	122:	(* manual down *)
		MD := TRUE;
		MU := FALSE;
		IF POS <= EXT_TRIG THEN
			(* extend cycle if bottom is reached *)
			POS := BYTE#0;
			last := tx;
			STATUS := BYTE#129;	(* extend *)
		END_IF;

	123:	(* auto positioning *)
		MD := rmp.DN;
		MU := rmp.UP;
		IF NOT (rmp.DN OR rmp.UP) THEN
			(* automatic position is reached *)
			IF POS <= EXT_TRIG THEN
				(* extend at bottom *)
				MD := TRUE;
				last := tx;
				STATUS := BYTE#129;	(* extend *)
			ELSIF POS >= USINT_TO_BYTE(USINT#255 - BYTE_TO_USINT(EXT_TRIG)) THEN
				(* extend at top *)
				MU := TRUE;
				last := tx;
				STATUS := BYTE#129;	(* extend *)
			ELSE
				STATUS := S_IN;
			END_IF;
		END_IF;

	124:	(* revert from top or bottom *)
		MD := rmp.DN;
		MU := rmp.UP;
		IF NOT(rmp.DN OR rmp.UP) THEN
(*		IF POS = rmp.IN THEN  *)
			PI_last := PI;
			STATUS := S_IN;
		END_IF;

	127:	(* lockout time *)
		IF (tx - last) >= T_LOCKOUT THEN
				STATUS := S_IN;
		END_IF;

	128:	(* calibration *)
		MU := TRUE;
		MD := FALSE;
		rmp.IN := BYTE#255;
		IF (tx - last) >= (T_UP +  T_EXT) THEN
			MU := FALSE;
			last := tx;
			STATUS := BYTE#127;	(* lockout *)
		END_IF;

	129: (* extend mode *)
		IF (tx - last) >= T_EXT THEN
			MU := FALSE;
			MD := FALSE;
			last := tx;
			STATUS := BYTE#127;	(* lockout *)
		END_IF;

ELSE
	MU := FALSE;
	MD := FALSE;
	IF PI <> PI_last THEN
		PI_last := PI;
		rmp.IN := PI;
		STATUS := BYTE#123;	(* auto positioning *)
	ELSIF POS = BYTE#0 AND RU THEN
		rmp.IN := R_POS_BOT;
		STATUS := BYTE#124;	(* revert *)
	ELSIF pos = BYTE#255 AND RD THEN
		rmp.IN := R_POS_TOP;
		STATUS := BYTE#124;	(* revert *)
	ELSE
		STATUS := S_IN;
	END_IF;
END_CASE;

(* From OSCAT LIBRARY, www.oscat.de *)
(* T_PLC_MS, _RMP_NEXT required *)
          
END_FUNCTION_BLOCK

FUNCTION_BLOCK BLIND_INPUT
  VAR_INPUT
    POS : BYTE;
    ANG : BYTE;
    S1 : BOOL;
    S2 : BOOL;
    IN : BOOL;
    PI : BYTE;
    AI : BYTE;
    SINGLE_SWITCH : BOOL;
    CLICK_EN : BOOL := TRUE;
    CLICK_TIME : TIME := t#500ms;
    MAX_RUNTIME : TIME := t#60s;
    MANUAL_TIMEOUT : TIME := t#1h;
    DEBOUNCE_TIME : TIME := t#20ms;
    DBL_CLK1 : BOOL := FALSE;
    DBL_POS1 : BYTE;
    DBL_ANG1 : BYTE;
    DBL_CLK2 : BOOL := FALSE;
    DBL_POS2 : BYTE := 255;
    DBL_ANG2 : BYTE := 255;
    D1_TOGGLE : BOOL := TRUE;
    D2_TOGGLE : BOOL := TRUE;
    MASTER_MODE : BOOL;
  END_VAR
  VAR_OUTPUT
    QU : BOOL := TRUE;
    QD : BOOL := TRUE;
    STATUS : BYTE;
    PO : BYTE := 255;
    AO : BYTE := 255;
    D1 : BOOL;
    D2 : BOOL;
  END_VAR
  VAR
    s1e : TOF;
    s2e : TOF;
    s1d : CLICK_MODE;
    s2d : CLICK_MODE;
    dir : BOOL;
    tx : TIME;
    last : TIME;
  END_VAR

            tx:= UDINT_TO_TIME(T_PLC_MS(en:=true));

(* inputs S1 and S2 are debounced and then decoded for multiple clicks *)
s1e(in := S1, pt := DEBOUNCE_TIME);
s2e(in := S2, pt := DEBOUNCE_TIME);
s1d(in := (s1e.Q AND NOT SINGLE_SWITCH) OR (s1e.Q AND SINGLE_SWITCH AND dir), t_long := CLICK_TIME);
s2d(in := (s2e.Q AND NOT SINGLE_SWITCH) OR (s1e.Q AND SINGLE_SWITCH AND NOT dir), t_long := CLICK_TIME);

(* if d1 and d2 are not toggle clear them to make sure they are only active for oine cycle *)
IF NOT d1_toggle THEN d1 := FALSE; END_IF;
IF NOT d2_toggle THEN d2 := FALSE; END_IF;

(* decode actions *)
IF (s1d.LONG AND s2d.LONG) OR (status = BYTE#139) THEN
   status := BYTE#139;
   IF NOT (s1d.LONG OR s2d.LONG)  THEN status := BYTE#130; END_IF;
ELSIF s1d.tp_LONG THEN
	status := BYTE#132;
ELSIF s2d.tp_LONG THEN
	status := BYTE#133;
ELSIF  s1d.SINGLE THEN
	IF click_en THEN
		(* if running then we stop otherwise start new direction *)
		IF QU XOR QD THEN
			status := BYTE#131;
		ELSE
			status := BYTE#134;
			last := tx;
			dir := NOT dir;
		END_IF;
	END_IF;
ELSIF  s2d.SINGLE THEN
	IF click_en THEN
		(* if running then we stop otherwise start new direction *)
		IF QU XOR QD THEN
			status := BYTE#131;
		ELSE
			status := BYTE#135;
			last := tx;
			dir := NOT dir;
		END_IF;
	END_IF;
ELSIF in THEN
	status := BYTE#136;
	last := tx;
ELSIF s1d.DOUBLE THEN
	IF dbl_clk1 THEN
		(* a position need to be set for a double click on S1 *)
		status := BYTE#137;
		last := tx;
	ELSE
		(* toggle the output when dbl_clk1 is not active *)
		D1 := NOT D1;
	END_IF;
ELSIF s2d.DOUBLE THEN
	IF dbl_clk2 THEN
		(* a position need to be set for a double click on S2 *)
		status := BYTE#138;
		last := tx;
	ELSE
		(* toggle the output when dbl_clk2 is not active *)
		(* in single switch mode we need to toggle d1 instead of d2 *)
		IF single_switch THEN D1 := NOT D1; ELSE D2 := NOT D2; END_IF;
	END_IF;
END_IF;


(* state machine *)
CASE BYTE_TO_INT(status) OF
	0:		(* power up operation *)
			status := BYTE#130;

	130:	(* automatic operation standby *)
			IF NOT master_mode THEN
				PO := POS;
				AO := ANG;
			END_IF;
			QU := TRUE;
			QD := TRUE;

	131:	(* manual operation standby *)
			QU := FALSE;
			QD := FALSE;
			PO := POS;
			AO := ANG;
			(* manual mode will be ended when timeout is reached *)
			IF tx - last >= manual_timeout THEN
				status := BYTE#130;
			END_IF;

	132:	(* manual operation up *)
			QU := TRUE;
			QD := FALSE;
			PO := POS; AO := ANG;
			last := tx;
			IF NOT s1d.LONG THEN status := BYTE#131; dir := NOT dir; END_IF;

	133:	(* manual operation down *)
			QU := FALSE;
			QD := TRUE;
			PO := POS; AO := ANG;
			last := tx;
			IF NOT s2d.LONG THEN	status := BYTE#131; dir := NOT dir; END_IF;

	134:	(* manual operation single click up *)
			QU := TRUE;
			QD := FALSE;
			PO := POS; AO := ANG;
			IF tx - last >= max_runtime THEN status := BYTE#131; END_IF;

	135:	(* manual operation single click dn *)
			QU := FALSE;
			QD := TRUE;
			PO := POS; AO := ANG;
			IF tx - last >= max_runtime THEN status := BYTE#131;	END_IF;

	136:	(* forced input in = true *)
			QU := TRUE;
			QD := TRUE;
			PO := PI; AO := AI;
			IF tx-last >= max_runtime THEN status := BYTE#130; END_IF;

	137:	(* double click1 position *)
			QU := TRUE;
			QD := TRUE;
			PO := DBL_POS1;
			AO := DBL_ANG1;
			IF tx - last >= max_runtime THEN status := BYTE#131; END_IF;

	138:	(* double click2 position *)
			QU := TRUE;
			QD := TRUE;
			PO := DBL_POS2;
			AO := DBL_ANG2;
			IF tx - last >= max_runtime THEN status := BYTE#131; END_IF;

	   139:   (* manual operation standby *)
	         QU := FALSE;
	         QD := FALSE;
	         PO := POS;
	         AO := ANG;

END_CASE;

(* From OSCAT LIBRARY, www.oscat.de *)
(* T_PLC_MS required *)
          
END_FUNCTION_BLOCK

FUNCTION_BLOCK BLIND_NIGHT
  VAR_INPUT
    UP : BOOL;
    DN : BOOL;
    S_IN : BYTE;
    PI : BYTE;
    AI : BYTE;
    E_NIGHT : BOOL := TRUE;
    E_DAY : BOOL := TRUE;
    DTIN : UDINT;
    SUNRISE : UDINT;
    SUNSET : UDINT;
    SUNRISE_OFFSET : TIME;
    SUNSET_OFFSET : TIME;
    NIGHT_POSITION : BYTE;
    NIGHT_ANGLE : BYTE;
  END_VAR
  VAR_OUTPUT
    QU : BOOL;
    QD : BOOL;
    STATUS : BYTE;
    PO : BYTE;
    AO : BYTE;
  END_VAR
  VAR
    night : BOOL;
    last_night : UDINT;
    last_day : UDINT;
  END_VAR

            IF NOT (up AND dn) AND night THEN
	(* manual operation at night will cancel operation for one night *)
	night := FALSE;
ELSIF (_DT_TO_TOD(dtin) > sunset + TIME_TO_UDINT(sunset_offset)) AND (last_night < _DT_TO_DATE(dtin)) AND NOT night AND e_night THEN
	(* enable night *)
	night := TRUE;
	last_night := _DT_TO_DATE(dtin);
ELSIF (_DT_TO_TOD(dtin) > sunrise + TIME_TO_UDINT(sunrise_offset)) AND (last_day < _DT_TO_DATE(dtin)) AND night AND e_day AND (last_night < _DT_TO_DATE(dtin)) THEN
	(* disable night *)
	night := FALSE;
	last_day := _DT_TO_DATE(dtin);
END_IF;

(* shade at night only in auto mode and enable = true *)
IF UP AND DN AND night THEN
	status := BYTE#141;
	po := night_position;
	ao := night_angle;
ELSE
	QU := UP;
	QD := DN;
	po := pi;
	ao := ai;
	status := s_in;
END_IF;

(* From OSCAT LIBRARY, www.oscat.de *)
          
END_FUNCTION_BLOCK

FUNCTION_BLOCK BLIND_SECURITY
  VAR_INPUT
    UP : BOOL;
    DN : BOOL;
    S_IN : BYTE;
    PI : BYTE;
    AI : BYTE;
    FIRE : BOOL;
    WIND : BOOL;
    ALARM : BOOL;
    DOOR : BOOL;
    RAIN : BOOL;
    ALARM_UP : BOOL := TRUE;
    WIND_UP : BOOL := TRUE;
    RAIN_UP : BOOL := TRUE;
    QU : BOOL;
    QD : BOOL;
    STATUS : BYTE;
    PO : BYTE;
    AO : BYTE;
  END_VAR

            IF Fire THEN

	QU := TRUE;

	QD := FALSE;

	status := BYTE#111;

ELSIF Wind THEN

	QU := Wind_up;

	QD := NOT wind_up;

	status := BYTE#112;

ELSIF alarm THEN

	QU := Alarm_up;

	QD := NOT Alarm_up;

	status := BYTE#113;

ELSIF Door THEN

	QU := TRUE;

	QD := FALSE;

	status := BYTE#114;

ELSIF Rain AND NOT (up XOR dn) THEN

	QU := rain_up;

	QD := NOT rain_up;

	status := BYTE#115;

ELSE

	QU := UP;

	QD := DN;

	status := S_IN;

	po := pi;

	ao := ai;

END_IF;


(* From OSCAT Library, www.OSCAT.de *)
          
END_FUNCTION_BLOCK

FUNCTION_BLOCK BLIND_SET
  VAR_INPUT
    UP : BOOL;
    DN : BOOL;
    S_IN : BYTE;
    PI : BYTE;
    AI : BYTE;
    PX : BYTE;
    AX : BYTE;
    IN : BOOL;
    OVERRIDE_MANUAL : BOOL;
    RESTORE_POSITION : BOOL;
    RESTORE_TIME : TIME := t#60s;
  END_VAR
  VAR_OUTPUT
    QU : BOOL;
    QD : BOOL;
    STATUS : BYTE;
    PO : BYTE;
    AO : BYTE;
  END_VAR
  VAR
    tx : TIME;
    last : TIME;
    ps : BYTE;
    as : BYTE;
  END_VAR

            tx:= UDINT_TO_TIME(T_PLC_MS(en:=true));

(* check inputs *)

IF IN THEN

	IF override_manual OR (UP AND DN) THEN

		status := 178;

	END_IF;

END_IF;



(* state machine *)

CASE byte_to_int(STATUS) OF

	0: (* power on state *)

		status := S_IN;



	178: (* force values from PX and AX *)

		PO := PX;

		AO := AX;

		QU := TRUE;

		QD := TRUE;

		(* check for end of forced position *)

		IF NOT in THEN

			STATUS := SEL(RESTORE_POSITION, S_IN, 179);

			last := tx;

		END_IF;



	179: (* restore previous position *)

		PO := ps;

		AO := as;

		IF ((PO = PI) AND (AO = AI))  OR tx - last >= RESTORE_TIME THEN

			status := S_IN;

		END_IF;



ELSE

	(* no operation transfer inputs to outputs *)

	PO := PI;

	ps := PI;

	AO := AI;

	as := AI;

	STATUS := S_IN;

	QU := UP;

	QD := DN;

END_CASE;




(* From OSCAT Library, www.OSCAT.de *)
          
END_FUNCTION_BLOCK

FUNCTION_BLOCK BLIND_SHADE
  VAR_INPUT
    UP : BOOL;
    DN : BOOL;
    PI : BYTE;
    AI : BYTE;
    S_IN : BYTE;
    ENABLE : BOOL;
    SUN : BOOL;
    SUNRISE_OFFSET : TIME := t#1h;
    SUNSET_PRESET : TIME := t#1h;
    SHADE_DELAY : TIME := t#60s;
    SHADE_POS : BYTE;
    DIRECTION : REAL := 180.0;
    ANGLE_OFFSET : REAL := 80.0;
    SLAT_WIDTH : REAL := 80.0;
    SLAT_SPACING : REAL := 60.0;
  END_VAR
  VAR_OUTPUT
    QU : BOOL;
    QD : BOOL;
    STATUS : BYTE;
    PO : BYTE;
    AO : BYTE;
  END_VAR
  VAR_IN_OUT
    CX : OSCAT_CALENDAR;
  END_VAR
  VAR
    sun_delay : TOF;
    angle : REAL;
  END_VAR

            (* the input sun is sent through tof which will delay the shade for the time shade_delay *)

sun_delay(IN := sun, PT := shade_delay);



IF UP AND DN AND enable AND sun_delay.Q AND cx.SUN_HOR > direction - angle_offset AND cx.SUN_HOR < direction + angle_offset AND

	_DT_TO_TOD(cx.UTC) > cx.SUN_RISE + TIME_TO_UDINT(sunrise_offset) AND _DT_TO_TOD(cx.UTC) < cx.SUN_SET - TIME_TO_UDINT(sunset_preset) THEN

	status := BYTE#151;

	QU := UP;

	QD := DN;

	(* position is predefined *)

	po := shade_pos;

	(* shading is active now calculate the slat angle *)

	(* calculate the max angle for the blind *)

	angle := DEG(ATAN(slat_spacing / slat_width));

	(* check if sun angle is between 0 and max angle *)

	IF cx.SUN_VER > 0.0 AND cx.SUN_VER < angle THEN

		angle := cx.SUN_VER + DEG(ACOS(COS(RAD(cx.SUN_VER))*slat_spacing / Slat_width));

		ao := INT_TO_BYTE(LIMIT(0,UDINT_TO_INT(TRUNC(angle * 2.833333333)), 255));

	ELSE

		ao := BYTE#255;

	END_IF;

ELSE

	QU := UP;

	QD := DN;

	po := pi;

	ao := ai;

	status := S_IN;

END_IF;




(* From OSCAT Library, www.OSCAT.de *)
          
END_FUNCTION_BLOCK

CONFIGURATION Config0
  RESOURCE Res0 ON PLC
    TASK task0(INTERVAL := T#20ms, PRIORITY := 0);
    PROGRAM instance0 WITH task0 : program0;
  END_RESOURCE
END_CONFIGURATION
